# EPICS autosave request: autosave/galil_motor_extras.req
$(P)$(M)_ESTALLTIME_SP
$(P)$(M)_STEPSMOOTH_SP
$(P)$(M)_UINDEX_CMD
$(P)$(M)_USWITCH_CMD
$(P)$(M)_USERDATADEADB_SP
$(P)$(M)_JAH_CMD
$(P)$(M)_JAHV_SP
$(P)$(M)_EGUAFTLIMIT_SP
$(P)$(M)_SSIINPUT_CMD
$(P)$(M)_SSITOTBITS_SP
$(P)$(M)_SSISINGLETBITS_SP
$(P)$(M)_SSIERRBITS_SP
$(P)$(M)_SSITIME_SP
$(P)$(M)_SSIDATA_CMD
$(P)$(M)_ECATADDR_SP
$(P)$(M)_ECATFLTRST_CMD
$(P)$(M)_BISSSTAT_POLL_CMD
$(P)$(M)_BISSINPUT_CMD
$(P)$(M)_BISSDATA1_SP
$(P)$(M)_BISSDATA2_SP
$(P)$(M)_BISSZP_SP
$(P)$(M)_BISSCD_SP
$(P)$(M)_BISSLEVEL_CMD
$(P)$(M)_STATUS_POLL_DELAY_CMD
$(P)$(M)_HOMEALLOWED_CMD
$(P)$(M)_STOPDELAY_SP
$(P)$(M)_AMPGAIN_CMD
$(P)$(M)_AMPCLGAIN_CMD
$(P)$(M)_AMPLC_SP
$(P)$(M)_ERRLIMIT_SP
$(P)$(M)_OFFONERR_CMD
$(P)$(M)_MTRTYPE_CMD
$(P)$(M)_MENCTYPE_CMD
$(P)$(M)_AENCTYPE_CMD
$(P)$(M)_WLP_CMD
$(P)$(M)_AUTOONOFF_CMD
$(P)$(M)_ONDELAY_SP
$(P)$(M)_OFFDELAY_SP
# $(P)$(M)_BRAKE_CMD
$(P)$(M)_AUTOBRAKE_CMD
$(P)$(M)_BRAKEPORT_SP
$(P)$(M)_BRAKEONDELAY_SP
$(P)$(M)_LIMITDISABLE_CMD
$(P)$(M)_ON_CMD
